// TIA Portal V18 export
VAR_GLOBAL   // PLC tag table "DQ"
   out_BeaconGreen AT %Q0.0 : Bool;
   out_BeaconRed AT %Q0.1 : Bool;
   out_BeaconYellow AT %Q0.2 : Bool;
   out_GenPallet AT %Q0.3 : Bool;
   out_GenBox AT %Q0.4 : Bool;
   out_5 AT %Q0.5 : Bool;
   out_6 AT %Q0.6 : Bool;
   out_7 AT %Q0.7 : Bool;
   out_8 AT %Q1.0 : Bool;
   out_Cov_0 AT %Q1.1 : Bool;
   out_Cov_1 AT %Q1.2 : Bool;
   out_Cov_2 AT %Q1.3 : Bool;
   out_Cov_3 AT %Q1.4 : Bool;
   out_Cov_4 AT %Q1.5 : Bool;
   out_Cov_5 AT %Q1.6 : Bool;
   out_15 AT %Q1.7 : Bool;
   out_Picker AT %Q2.0 : Bool;
   out_17 AT %Q2.1 : Bool;
   out_18 AT %Q2.2 : Bool;
   out_19 AT %Q2.3 : Bool;
   out_20 AT %Q2.4 : Bool;
   out_21 AT %Q2.5 : Bool;
   out_22 AT %Q2.6 : Bool;
   out_23 AT %Q2.7 : Bool;
   out_BladesFroward AT %Q28.0 : Bool;
   out_BladesBackward AT %Q28.1 : Bool;
   out_26 AT %Q28.2 : Bool;
   out_27 AT %Q28.3 : Bool;
END_VAR
